// Mitsubishi GX Works2 project: 气路版本2   PLC: FX2N/FX2NC

PROGRAM MAIN
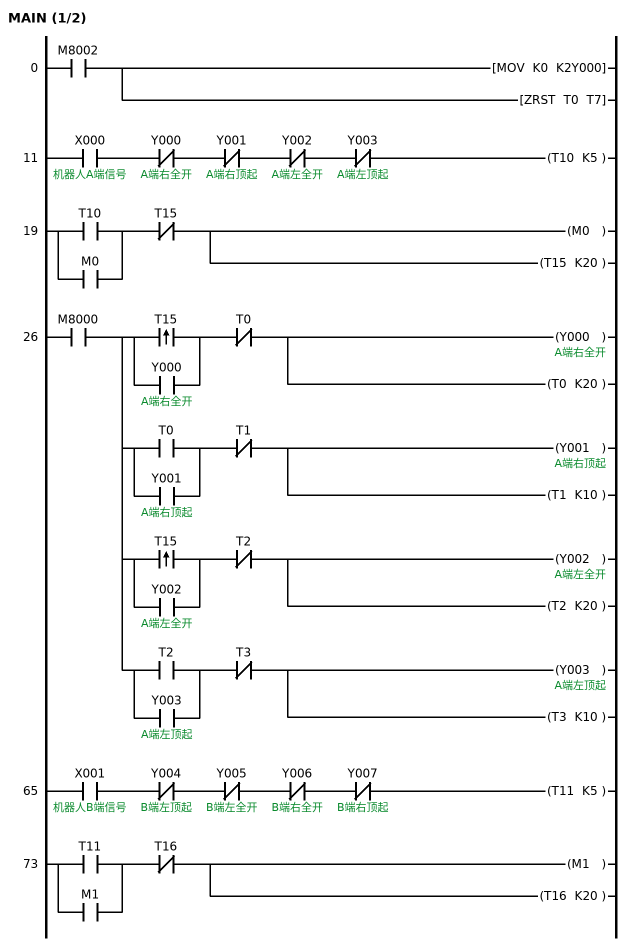
0     LD      M8002
      MOV     K0 K2Y000  ; A端右全开
      ZRST    T0 T7
11    LD      X000  ; 机器人A端信号
      ANI     Y000  ; A端右全开
      ANI     Y001  ; A端右顶起
      ANI     Y002  ; A端左全开
      ANI     Y003  ; A端左顶起
      OUT     T10 K5
19    LD      T10
      OR      M0
      ANI     T15
      OUT     M0
      OUT     T15 K20
26    LD      M8000
      MPS
      LDP     T15
      OR      Y000  ; A端右全开
      ANB
      ANI     T0
      OUT     Y000  ; A端右全开
      OUT     T0 K20
      MRD
      LD      T0
      OR      Y001  ; A端右顶起
      ANB
      ANI     T1
      OUT     Y001  ; A端右顶起
      OUT     T1 K10
      MRD
      LDP     T15
      OR      Y002  ; A端左全开
      ANB
      ANI     T2
      OUT     Y002  ; A端左全开
      OUT     T2 K20
      MPP
      LD      T2
      OR      Y003  ; A端左顶起
      ANB
      ANI     T3
      OUT     Y003  ; A端左顶起
      OUT     T3 K10
65    LD      X001  ; 机器人B端信号
      ANI     Y004  ; B端左顶起
      ANI     Y005  ; B端左全开
      ANI     Y006  ; B端右全开
      ANI     Y007  ; B端右顶起
      OUT     T11 K5
73    LD      T11
      OR      M1
      ANI     T16
      OUT     M1
      OUT     T16 K20
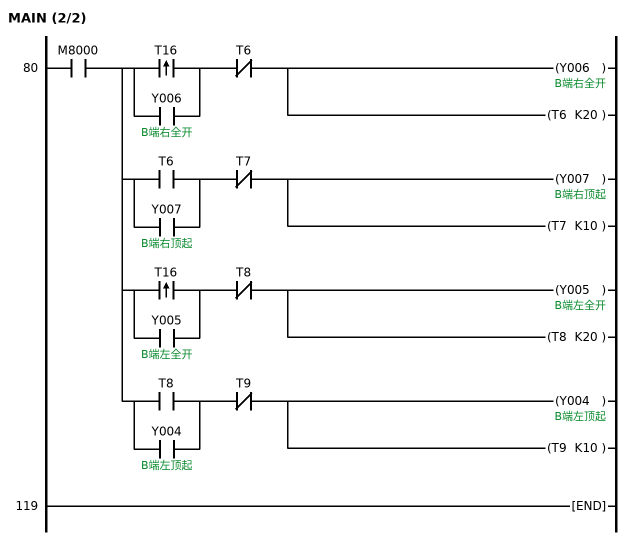
80    LD      M8000
      MPS
      LDP     T16
      OR      Y006  ; B端右全开
      ANB
      ANI     T6
      OUT     Y006  ; B端右全开
      OUT     T6 K20
      MRD
      LD      T6
      OR      Y007  ; B端右顶起
      ANB
      ANI     T7
      OUT     Y007  ; B端右顶起
      OUT     T7 K10
      MRD
      LDP     T16
      OR      Y005  ; B端左全开
      ANB
      ANI     T8
      OUT     Y005  ; B端左全开
      OUT     T8 K20
      MPP
      LD      T8
      OR      Y004  ; B端左顶起
      ANB
      ANI     T9
      OUT     Y004  ; B端左顶起
      OUT     T9 K10
119   END
END_PROGRAM
